FUNCTION_BLOCK FB_BA_2WayButton_IO EXTENDS FB_BA_VIEW
VAR_INPUT
END_VAR
VAR_INPUT CONSTANT
	Swi1					: FB_BA_BI_IO;		
	Swi2					: FB_BA_BI_IO;		
END_VAR
VAR_OUTPUT
	bPresentValue1			: BOOL;	
	bPresentValue2			: BOOL;	
END_VAR
VAR
END_VAR

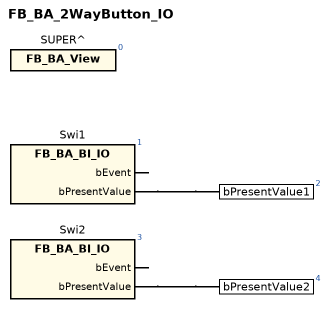
SUPER^(); // FB_BA_View
Swi1(); // FB_BA_BI_IO
bPresentValue1 := Swi1.bPresentValue;
Swi2(); // FB_BA_BI_IO
bPresentValue2 := Swi2.bPresentValue;

METHOD FB_init : BOOL
VAR_INPUT
	bInitRetains : BOOL; // if TRUE, the retain variables are initialized (warm start / cold start)
	bInCopyCode : BOOL;  // if TRUE, the instance afterwards gets moved into the copy code (online change)
END_VAR
Swi1.iParent					:= THIS^;
Swi1.iLabel						:= LblUniFieldDevice.SensorButton_Input;	
Swi1.sObjectName				:= '{Idx=01}';	
Swi1.sDeviceType				:= '';
Swi1.bEnOutOfService			:= FALSE;
Swi1.ePolarity					:= E_BA_Polarity.eNormal;
Swi1.sActiveText 				:= Texts.txtOn;
Swi1.sInactiveText 				:= Texts.txtOff;
Swi1.nStateChangeCount			:= 0;
Swi1.nActiveTimeElapsed			:= 0;
Swi1.nEventClassID				:= EventClasses.NotificationSimple;
Swi1.stTimeDelay.nToNormal		:= BA2_Param.nDefTimeDelay_ToNormal;
Swi1.stTimeDelay.nToAbnormal	:= BA2_Param.nDefTimeDelay_ToAbnormal;
Swi1.bAlarmValue				:= TRUE;
Swi1.bAcknowledgeRm				:= FALSE;		
Swi1.aEventTransitionText[1]	:= Texts.txtOff;
Swi1.aEventTransitionText[2]	:= Texts.txtNone;
Swi1.aEventTransitionText[3]	:= Texts.txtOn;
Swi1.bEventDetectionEnable		:= FALSE;
Swi1.eEnPlantLock				:= E_BA_LockPriority.eNoLock;	

Swi2.iParent					:= THIS^;
Swi2.iLabel						:= LblUniFieldDevice.SensorButton_Input;	
Swi2.sObjectName				:= '{Idx=02}';	
Swi2.sDeviceType				:= '';
Swi2.bEnOutOfService			:= FALSE;
Swi2.ePolarity					:= E_BA_Polarity.eNormal;
Swi2.sActiveText 				:= Texts.txtOn;
Swi2.sInactiveText 				:= Texts.txtOff;
Swi2.nStateChangeCount			:= 0;
Swi2.nActiveTimeElapsed			:= 0;
Swi2.nEventClassID				:= EventClasses.NotificationSimple;
Swi2.stTimeDelay.nToNormal		:= BA2_Param.nDefTimeDelay_ToNormal;
Swi2.stTimeDelay.nToAbnormal	:= BA2_Param.nDefTimeDelay_ToAbnormal;
Swi2.bAlarmValue				:= TRUE;
Swi2.bAcknowledgeRm				:= FALSE;		
Swi2.aEventTransitionText[1]	:= Texts.txtOff;
Swi2.aEventTransitionText[2]	:= Texts.txtNone;
Swi2.aEventTransitionText[3]	:= Texts.txtOn;
Swi2.bEventDetectionEnable		:= FALSE;
Swi2.eEnPlantLock				:= E_BA_LockPriority.eNoLock;
END_METHOD

END_FUNCTION_BLOCK

(* stored: Version 1.1.0.1, ProductVersion 3.1.4024.6
   POU FB_BA_2WayButton_IO: Id {3dbe968e-87cf-49df-99fd-5e696ba9a413}, SpecialFunc None
   Method FB_init: Id {cc5b5b4c-5563-47a7-af0b-dd55ebace0bc} *)
